(* PLC project model, Beckhoff Automation Beckhoff MLlib 3.1.251201.0 *)
(* stored: creationDateTime 2026-07-10T12:15:33.6636674, modificationDateTime 2026-07-10T12:15:33.6636674 *)

TYPE ST_modelInput :
STRUCT

	{attribute 'hide'} _header_DO_NOT_CHANGE : ARRAY[0..63] OF SINT := [-1,-112,120,86,52,18,-1,-1,1,-1,0,0,-1,-1,-112,-112,55,-22,8,-62,15,-11,-53,-120,-65,-26,40,-59,-103,80,20,5,37,-41,0,-16,-125,-33,-67,117,-59,70,-31,-53,-46,-33,-68,-19,80,2,0,0,0,0,0,0,0,0,0,0,0,0,0,0];
	in_input_tensor : ARRAY[0..0,0..32,0..3] OF REAL;

END_STRUCT
END_TYPE

TYPE ST_modelOutput :
STRUCT

	{attribute 'hide'} _header_DO_NOT_CHANGE : ARRAY[0..63] OF SINT := [-1,-112,120,86,52,18,-1,-1,1,-1,0,0,-1,-1,-112,-112,65,64,108,85,118,21,-37,1,110,122,-102,19,93,-117,-35,-43,3,-45,33,-52,25,-24,90,7,83,36,22,5,-43,-65,-103,-61,76,0,0,0,0,0,0,0,0,0,0,0,0,0,0,0];
	out_prediction_tensor : ARRAY[0..0,0..2] OF REAL;

END_STRUCT
END_TYPE
